Universal Robots PolyScope program: RotateAroundAnAxis.urp

ProgramRoot directory=/home/ur/ursim-3.1/programs/FAQ/RotateAroundAnAxis; kinematics=(a=[0.00023, -0.38811, -0.39243, -0.00016, 0.00019, 0], d=[0.08925, 195.22769, -194.66383, -0.45311, 0.09509, 0.08264], alpha=[1.57049, -0.00089, 0.00686, 1.56999, -1.56996, 0], deltaTheta=[-0.00001, -0.41907, 0.4289, -6.29306, -0.00007, 0], status=notLinearised); lastSavedInVersion=(project__name=Polyscope, major__version=3, minor__version=1, svn__revision=16916, build__date=Feb 06 2015, 15:15:00); name=RotateAroundAnAxis; programVersion=(project__name=PolyScope, major__version=1, minor__version=0, svn__revision=0); robotEnvironmentFileName=RotateAroundAnAxis; serialNumberRobot=2014350001
  BeforeStart description=COMMAND_SEQUENCE_BEFORE_PROGRAM_START; name=BeforeStart
    Move cartesianAcceleration=1.2; cartesianSpeed=0.25; jointAcceleration=1.3962634015954636; jointSpeed=1.0471975511965976; sharedProcessMoveBlendRadius=0.025; motionType=JOINT_SPACE
      Waypoint blendRadius=0.05; cartesianAcceleration=1.2; cartesianSpeed=0.25; jointAcceleration=1.3962634015954636; jointSpeed=1.0471975511965976; nextMotionTime=2.0; stoppoint=true; useSharedBlendParameter=true; useSharedParameters=true; position=TCP in base x=-351.288 y=-433.897 z=317.217 mm, rx=1.2452 ry=2.2988 rz=-0.3855 rad; joints [34.751, -80.904, 99.482, -110.617, -56.625, 2.463] deg; positionType=RELATIVE_POSITION; waypointPoseInFeatureCoordinates=(pos=(x=-0.3512875326114385, y=-0.4338971767078812, z=0.3172165170741499), rot=(x=1.2452365150751565, y=2.2987621955204807, z=-0.38549480530047175)); name=Relative; relativeFromJointPositionVector=(joint=[0.60651, -1.41204, 1.73628, -1.93063, -0.9883, 0.04298], isUndefined=false); relativeFromToolAxisAngle=(x=1.245152784027271, y=2.298762027301543, z=-0.38554821387687904); relativeFromToolPosition=(x=-0.35126939034874455, y=-0.4339042942377807, z=0.31722733091517563)
      Waypoint blendRadius=0.05; cartesianAcceleration=1.2; cartesianSpeed=0.25; jointAcceleration=1.3962634015954636; jointSpeed=1.0471975511965976; nextMotionTime=2.0; stoppoint=true; useSharedBlendParameter=true; useSharedParameters=true; position=TCP in base x=-351.279 y=-433.902 z=317.238 mm, rx=1.2451 ry=2.2988 rz=-0.3856 rad; joints [34.751, -80.904, 99.482, -110.617, -56.625, 2.463] deg; positionType=FIXED_POSITION; waypointPoseInFeatureCoordinates=(pos=(x=-0.35127882959782314, y=-0.43390202451533194, z=0.3172379823648375), rot=(x=1.2451281537231513, y=2.298801117333702, z=-0.38558808795887145)); name=Home
      Suppressed suppressedNode=(PositionNode=(default=(blendRadius=0.02, cartesianAcceleration=1.2, cartesianSpeed=0.25, jointAcceleration=1.3962634015954636, jointSpeed=1.0471975511965976, nextMotionTime=2.0, specifyNextMotionTime=false, stoppoint=false, useSharedBlendParameter=false, useSharedParameters=true, positionType=FIXED_POSITION)), WaypointNode=(default=(name=Waypoint_1, relativeFromJointPositionVector=(joint=[nan, nan, nan, nan, nan, nan], isUndefined=true), relativeFromToolAxisAngle=(x=0.0, y=0.0, z=0.0), relativeFromToolPosition=(x=0.0, y=0.0, z=0.0))))
      Assignment expr=get_forward_kin(); operatorValueType=INTEGER; valueSource=EXPRESSION
      Assignment expr=p[0,0,0.1,0,0,0]; operatorValueType=INTEGER; valueSource=EXPRESSION
      Assignment expr=p[0,0,0,d2r(45),0,0]; operatorValueType=INTEGER; valueSource=EXPRESSION
      Assignment expr=p[0,0,0,-d2r(45),0,0]; operatorValueType=INTEGER; valueSource=EXPRESSION
      Assignment expr=p[0,0,0,0,d2r(45),0]; operatorValueType=INTEGER; valueSource=EXPRESSION
      Assignment expr=p[0,0,0,0,-d2r(45),0]; operatorValueType=INTEGER; valueSource=EXPRESSION
      Assignment expr=p[0,0,0,0,0,d2r(60)]; operatorValueType=INTEGER; valueSource=EXPRESSION
      Assignment expr=p[0,0,0,0,0,-d2r(60)]; operatorValueType=INTEGER; valueSource=EXPRESSION
      Folder name=Calculate XYZ
        Assignment expr=pose_add(ExpressionVariableNode,ExpressionVariableNode); operatorValueType=INTEGER; valueSource=EXPRESSION
        Assignment expr=pose_trans(ExpressionVariableNode,ExpressionVariableNode); operatorValueType=INTEGER; valueSource=EXPRESSION
      Folder name=Calculate Base Coordinate
        Assignment expr=pose_add(ExpressionVariableNode,ExpressionVariableNode); operatorValueType=INTEGER; valueSource=EXPRESSION
        Assignment expr=pose_add(ExpressionVariableNode,ExpressionVariableNode); operatorValueType=INTEGER; valueSource=EXPRESSION
        Assignment expr=pose_add(ExpressionVariableNode,ExpressionVariableNode); operatorValueType=INTEGER; valueSource=EXPRESSION
        Assignment expr=pose_add(ExpressionVariableNode,ExpressionVariableNode); operatorValueType=INTEGER; valueSource=EXPRESSION
        Assignment expr=pose_add(ExpressionVariableNode,ExpressionVariableNode); operatorValueType=INTEGER; valueSource=EXPRESSION
        Assignment expr=pose_add(ExpressionVariableNode,ExpressionVariableNode); operatorValueType=INTEGER; valueSource=EXPRESSION
      Folder name=Calculate Tool Coordinate
        Assignment expr=pose_trans(ExpressionVariableNode,ExpressionVariableNode); operatorValueType=INTEGER; valueSource=EXPRESSION
        Assignment expr=pose_trans(ExpressionVariableNode,ExpressionVariableNode); operatorValueType=INTEGER; valueSource=EXPRESSION
        Assignment expr=pose_trans(ExpressionVariableNode,ExpressionVariableNode); operatorValueType=INTEGER; valueSource=EXPRESSION
        Assignment expr=pose_trans(ExpressionVariableNode,ExpressionVariableNode); operatorValueType=INTEGER; valueSource=EXPRESSION
        Assignment expr=pose_trans(ExpressionVariableNode,ExpressionVariableNode); operatorValueType=INTEGER; valueSource=EXPRESSION
        Assignment expr=pose_trans(ExpressionVariableNode,ExpressionVariableNode); operatorValueType=INTEGER; valueSource=EXPRESSION
  MainProgram cartesianAcceleration=1.2; cartesianSpeed=0.25; jointAcceleration=1.3962634015954636; jointSpeed=1.0471975511965976; sharedProcessMoveBlendRadius=0.0; motionType=JOINT_SPACE
    Move cartesianAcceleration=1.2; cartesianSpeed=0.25; jointAcceleration=1.3962634015954636; jointSpeed=1.0471975511965976; sharedProcessMoveBlendRadius=0.025; motionType=CARTESIAN_SPACE
      Folder name=Move Around Base Coordinate
        Folder name=pose_add
          While count=3; type=LOOP_COUNT
            Waypoint blendRadius=0.05; cartesianAcceleration=1.2; cartesianSpeed=0.25; jointAcceleration=1.3962634015954636; jointSpeed=1.0471975511965976; nextMotionTime=2.0; stoppoint=true; useSharedBlendParameter=true; useSharedParameters=true; positionType=VARIABLE_POSITION; name=Pos_1
            Waypoint blendRadius=0.05; cartesianAcceleration=1.2; cartesianSpeed=0.25; jointAcceleration=1.3962634015954636; jointSpeed=1.0471975511965976; nextMotionTime=2.0; stoppoint=true; useSharedBlendParameter=true; useSharedParameters=true; positionType=VARIABLE_POSITION; name=Pos_1
      Folder name=Move Around Tool Coordinate
        Folder name=pose_trans
          While count=3; type=LOOP_COUNT
            Waypoint blendRadius=0.05; cartesianAcceleration=1.2; cartesianSpeed=0.25; jointAcceleration=1.3962634015954636; jointSpeed=1.0471975511965976; nextMotionTime=2.0; stoppoint=true; useSharedBlendParameter=true; useSharedParameters=true; positionType=VARIABLE_POSITION; name=Pos_1
            Waypoint blendRadius=0.05; cartesianAcceleration=1.2; cartesianSpeed=0.25; jointAcceleration=1.3962634015954636; jointSpeed=1.0471975511965976; nextMotionTime=2.0; stoppoint=true; useSharedBlendParameter=true; useSharedParameters=true; positionType=VARIABLE_POSITION; name=Pos_1
      Folder name=Rotate Around Base Coordinate
        Suppressed 
        Suppressed 
        Folder name=pose_add RZ
          While count=3; type=LOOP_COUNT
            Waypoint blendRadius=0.05; cartesianAcceleration=1.2; cartesianSpeed=0.25; jointAcceleration=1.3962634015954636; jointSpeed=1.0471975511965976; nextMotionTime=2.0; stoppoint=true; useSharedBlendParameter=true; useSharedParameters=true; positionType=VARIABLE_POSITION; name=Pos_1
            Waypoint blendRadius=0.05; cartesianAcceleration=1.2; cartesianSpeed=0.25; jointAcceleration=1.3962634015954636; jointSpeed=1.0471975511965976; nextMotionTime=2.0; stoppoint=true; useSharedBlendParameter=true; useSharedParameters=true; positionType=VARIABLE_POSITION; name=Pos_1
            Waypoint blendRadius=0.05; cartesianAcceleration=1.2; cartesianSpeed=0.25; jointAcceleration=1.3962634015954636; jointSpeed=1.0471975511965976; nextMotionTime=2.0; stoppoint=true; useSharedBlendParameter=true; useSharedParameters=true; positionType=VARIABLE_POSITION; name=Pos_1
      Folder name=Rotate Around Tool Coordinate
        Suppressed 
        Suppressed 
        Folder name=pose_trans RZ
          While count=3; type=LOOP_COUNT
            Waypoint blendRadius=0.05; cartesianAcceleration=1.2; cartesianSpeed=0.25; jointAcceleration=1.3962634015954636; jointSpeed=1.0471975511965976; nextMotionTime=2.0; stoppoint=true; useSharedBlendParameter=true; useSharedParameters=true; positionType=VARIABLE_POSITION; name=Pos_1
            Waypoint blendRadius=0.05; cartesianAcceleration=1.2; cartesianSpeed=0.25; jointAcceleration=1.3962634015954636; jointSpeed=1.0471975511965976; nextMotionTime=2.0; stoppoint=true; useSharedBlendParameter=true; useSharedParameters=true; positionType=VARIABLE_POSITION; name=Pos_1
            Waypoint blendRadius=0.05; cartesianAcceleration=1.2; cartesianSpeed=0.25; jointAcceleration=1.3962634015954636; jointSpeed=1.0471975511965976; nextMotionTime=2.0; stoppoint=true; useSharedBlendParameter=true; useSharedParameters=true; positionType=VARIABLE_POSITION; name=Pos_1
